// TIA Portal project "TEMPERATURE" (V16)

(* hardware
DEVICE "S7-1200 station_1"  S7-1200 Station
   slot 0: "Rack_0"  S7-1200 Rack  Rack  V1.0
   slot 1: "PLC_1"  CPU 1212C AC/DC/Rly  6ES7 212-1BE40-0XB0  V4.0
*)

// ===== PLC "PLC_1"  CPU 1212C AC/DC/Rly =====

VAR_GLOBAL   // PLC tag table "Default tag table"
   "K1" AT %Q0.0 : Bool;
   "stop1" AT %I0.4 : Bool;
   "k2" AT %Q0.1 : Bool;
   "X" AT %M0.0 : Bool;
   "K3" AT %Q0.2 : Bool;
   "start1" AT %I0.2 : Bool;
   "T1 tag" AT %M0.1 : Bool;
   "T1 tag(1)" AT %M0.2 : Bool;
   "T3 tag" AT %M0.3 : Bool;
   "Y" AT %M1.0 : Bool;
   "Z" AT %M1.2 : Bool;
   "Tag_1" AT %I0.3 : Bool;
   "sensor" AT %I0.6 : Bool;
   "delay 5S" AT %M0.4 : Bool;
   "SENSOR(1)" AT %I0.5 : Bool;
   "START" AT %I0.1 : Bool;
END_VAR

// folder: System blocks/Program resources

DATA_BLOCK "T1"   // DB2
{ S7_Optimized_Access := 'TRUE' }
AUTHOR : Simatic
FAMILY : IEC
NAME : IEC_TMR
VERSION : 1.0
// stored: InstanceOfName IEC_TIMER
"IEC_TIMER"
BEGIN
END_DATA_BLOCK

// folder: (top level)

ORGANIZATION_BLOCK "Main"   // OB1, LAD, ProgramCycle
TITLE = "Main Program Sweep (Cycle)"
{ S7_Optimized_Access := 'TRUE' }
VERSION : 0.1
   VAR_INPUT
      Initial_Call : Bool;   // Initial call of this OB
      Remanence : Bool;   // =True, if remanent data are available
   END_VAR
BEGIN

REGION Network 1: start
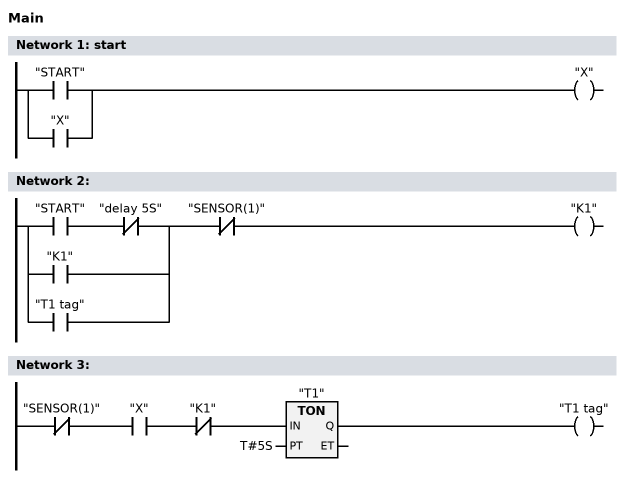
   RUNG wire#powerrail
      Contact( "START" )
      wire#w1
      Coil( "X" )
   END_RUNG
   RUNG wire#powerrail
      Contact( "X" )
   END_RUNG wire#w1
   // the same network as SCL:
   "X" := "START" OR "X";
END_REGION

REGION Network 2
   RUNG wire#powerrail
      Contact( "START" )
      I_Contact( "delay 5S" )
      wire#w1
      I_Contact( "SENSOR(1)" )
      Coil( "K1" )
   END_RUNG
   RUNG wire#powerrail
      Contact( "K1" )
   END_RUNG wire#w1
   RUNG wire#powerrail
      Contact( "T1 tag" )
   END_RUNG wire#w1
   // the same network as SCL:
   "K1" := (("START" AND NOT "delay 5S") OR "K1" OR "T1 tag") AND NOT "SENSOR(1)";
END_REGION

REGION Network 3
   "T1".TON(IN := NOT "SENSOR(1)" AND "X" AND NOT "K1", PT := T#5S);
   "T1 tag" := "T1".Q;
END_REGION
END_ORGANIZATION_BLOCK